// This function has been automatically generated from the project information.
{attribute 'signature_flag' := '1073741824'}
{attribute 'TcGenerated'}
{attribute 'no-analysis'}
FUNCTION F_GetTitle : WSTRING
VAR_INPUT
	
END_VAR

F_GetTitle := "FileIO";

END_FUNCTION

(* stored: Version 1.1.0.1
   POU F_GetTitle: Id {b7d02d0a-2197-46d6-a438-a29e5f9d8bee}, SpecialFunc None *)
